{attribute 'qualified_only'}
{attribute 'strict'}
TYPE E_MMVehicleInputType :
(
	eMMVehicleInputType_VehicleID			:= 0,	// MagneMotion ID
	eMMVehicleInputType_CarrierID			:= 1,	// RFID scanned ID from Carrier
	eMMVehicleInputType_LastID 				:= 2,	// RFID scanned Id from Last
	eMMVehicleInputType_ArticleID 			:= 3,
	eMMVehicleInputType_LastTypeID			:= 4,
	eMMVehicleInputType_StationID			:= 5,
	eMMVehicleInputType_CellID				:= 6,
	eMMVehicleInputType_EmptyVehicles		:= 7,
	eMMVehicleInputType_ReleasedVehicles	:= 8,
	eMMVehicleInputType_AllVehicles			:= 9
);
END_TYPE

(* stored: Version 1.1.0.1, ProductVersion 3.1.4024.5
   EnumerationTextList E_MMVehicleInputType: Id {ca9eeba8-1c9b-4181-ad08-f02832e25ced} *)
